TYPE AX5000_P_1005 :
STRUCT
	Debug_pointer_2_value:UDINT;
END_STRUCT
END_TYPE

(* stored: Version 1.1.0.1, ProductVersion 3.1.4024.3
   DUT AX5000_P_1005: Id {33ac19fb-3444-4306-a33f-c4de56d7cfe9} *)
